FUNCTION_BLOCK FB_LAMP_DIAG EXTENDS FB_LAMP_ONOFF IMPLEMENTS I_LampCtrl_Diag;
VAR_INPUT
END_VAR
VAR_OUTPUT
END_VAR
VAR
	iInTemperatureHw	AT %I*	: INT;
END_VAR

METHOD Diag : BOOL
Diag := FALSE;

IF iInTemperatureHw > 200 THEN
	SUPER^.OFF();
END_IF

DIAG := TRUE;
END_METHOD

END_FUNCTION_BLOCK

(* stored: Version 1.1.0.1, ProductVersion 3.1.4024.12
   POU FB_LAMP_DIAG: Id {59524f85-dde9-4bed-ba94-132faece4afc}, SpecialFunc None
   Method Diag: Id {64efed3b-e6da-4fa5-a978-5b15132c7a69} *)
